// This is a very ugly hack because I'm being lazy.
// I'm sure there is some better/more standard way.
FUNCTION_BLOCK FB_GetVacuumAMSID
VAR_INPUT
END_VAR
VAR_OUTPUT
	Busy : BOOL := TRUE;
	VacuumNetID : T_AmsNetID;
END_VAR
VAR
	DoCallOnce : BOOL := TRUE;
	DoOnce : BOOL := TRUE;
	GetLocalAMSId : FB_GetLocalAmsNetId;	

END_VAR
VAR_TEMP
	NetIDLen : INT;
END_VAR

(* We only really want to compute the netid once.
This requires performing the GetLocalAMSId call once and waiting for the result,
and then doing the processing of the result once. *)
IF NOT DoOnce AND NOT DoCallOnce THEN
	RETURN;
END_IF
GetLocalAMSId(bExecute :=  DoCallOnce, tTimeOut := T#5S);
DoCallOnce := FALSE ;
Busy := GetLocalAMSId.bBusy;
IF Busy THEN
	RETURN;
END_IF
IF DoOnce THEN
	DoOnce := FALSE;
	NetIDLen := LEN(GetLocalAMSId.AddrString);
	VacuumNetID := CONCAT(LEFT(GetLocalAMSId.AddrString, NetIDLen-4), '.3.1');
END_IF

END_FUNCTION_BLOCK

(* stored: Version 1.1.0.1, ProductVersion 3.1.4022.16
   POU FB_GetVacuumAMSID: Id {1d0d95ca-2f0a-4841-bf10-7d1e2b4b3cf2}, SpecialFunc None *)
